FUNCTION_BLOCK TestFuntionBlock
VAR
	nCounter : LINT;
	
END_VAR

nCounter := nCounter +1;

END_FUNCTION_BLOCK

(* stored: Version 1.1.0.1, ProductVersion 3.1.4024.9
   POU TestFuntionBlock: Id {b67aa33f-7126-40c2-946d-4429c73b2e3d}, SpecialFunc None *)
